Staubli VAL3: userPage.dtx

bool Show
public bool bListItemRef
bool bReadWrite[6]
  [0] = true
  [1] = true
  [2] = true
  [3] = true
  [4] = true
  [5] = true
public bool bShowDialog
public bool bUseEscape
public bool bUseRefresh = true
public num nBottomX[2]
  [0] = 15
  [1] = 15
public num nBottomY = 6
num nFirst
num nKey
num nOffSet
num nOldValue[2]
  [0] = 200
  [1] = 200
public num nPage = 100000
public num nParaAdjustType
num nTest
public num nToSuperV = -1
public num nTopX[2]
  [0] = 20
  [1] = 20
public num nTopY = 3
public num nView
public string sItems[6]
  [0] = "J1 :   5    "
  [1] = "J2 :  12    "
  [2] = "J3 : 104    "
  [3] = "J4 :  96    "
  [4] = "J5 :  60    "
  [5] = "J6 :-221    "
string sMessage = "是否删除该项?"
public string sTitle = "Home关节位置"
public string sToSuperV
string stest[11]
  [0] = "sbx"
  [1] = "sdfgsd"
  [2] = "bsfghsfh"
  [3] = "sdfgsdfg"
  [4] = "shsgh"
  [5] = "ghdfh"
  [6] = "snsfg"
  [7] = "sfgsg"
  [8] = "sfgsdfg"
  [9] = "sfgs"
  [10] = "dfsgs"
string stest2
string stest3
